TYPE EngStruct :
STRUCT
	uptime : STRING;
END_STRUCT
END_TYPE

(* stored: Version 1.1.0.1, ProductVersion 3.1.4024.10
   DUT EngStruct: Id {9c65b1a4-b473-4fba-b7fb-19a26602dbf4} *)
